ABB RobotStudio station: Sixth Assignment.rspag

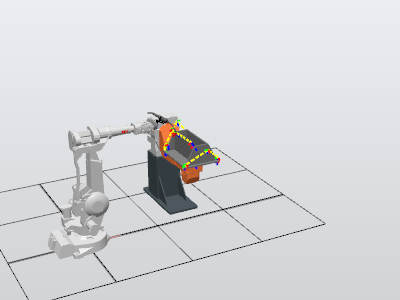
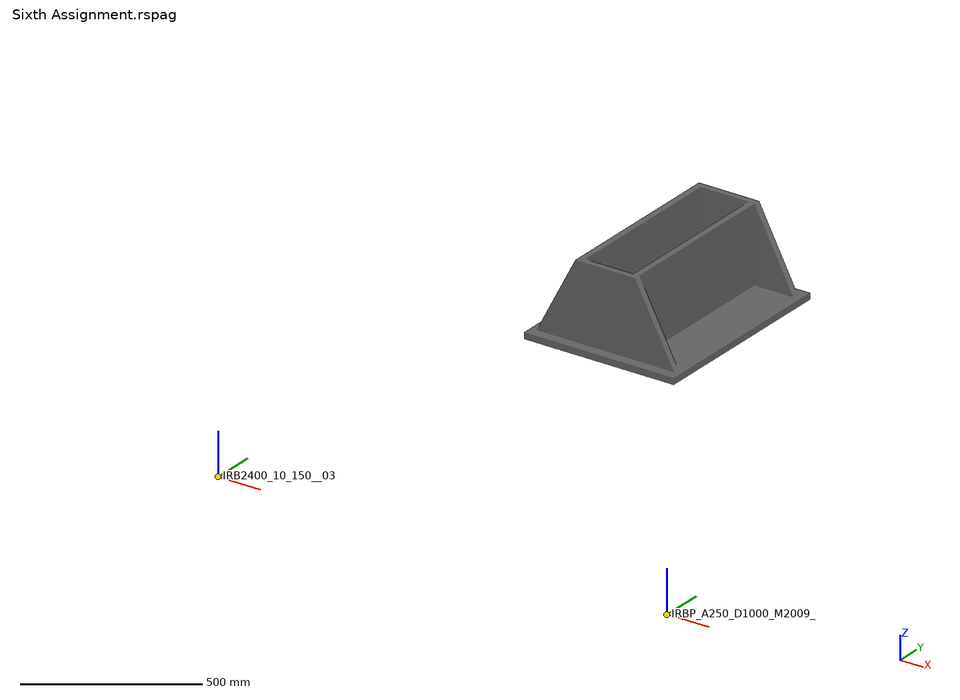
[picture v1: parts stored in the station drawn from their meshes, with robot base, taught points and paths (robot models come from the ABB library and are not in the file)]
--- station ---
Station station (saved by RobotStudio 24.1.10713.1)
Controller Controller
  mechanical unit ROB_1: IRB2400_10_150__03, 6 joints, base frame (0, 0, 0) mm
  mechanical unit STN1: IRBP_A250_D1000_M2009_REV1_01, 2 joints, base frame (0, 0, 0) mm
Layout (positions relative to the parent item):
  - IRB2400_10_150__03 [mechanism, from %ABB.RobotStudio.Models.IRB2400%\IRB2400_10_150_G_03.rslib] at (0, 0, 0) mm; joint values [0, 0.0266, 0.0287, -3.1416, -0.0726, 3.1416] (rad or m)
  - AW_Gun_PSF_25 [mechanism, from %ABB.RobotStudio.Models.ArcWelding%\AW_Gun_PSF_25.rslib] at (961.88, 0, 1424.46) mm, rotated rx 180 ry 84.2 rz 180 deg
  - IRBP_A250_D1000_M2009_REV1_01 [mechanism] at (1500, 0, 0) mm, rotated rx 0 ry 0 rz 90 deg; joint values [0, 0] (rad or m)
      links: Base, Link1, Link2
  - weldpiece [part] at (1500, 0, 900) mm, rotated rx 0 ry 0 rz -90 deg, size 650 x 500 x 270 mm
Attachment: AW_Gun_PSF_25 is attached to IRB2400_10_150__03 / Link6
Attachment: weldpiece is attached to IRBP_A250_D1000_M2009_REV1_01 / Link2

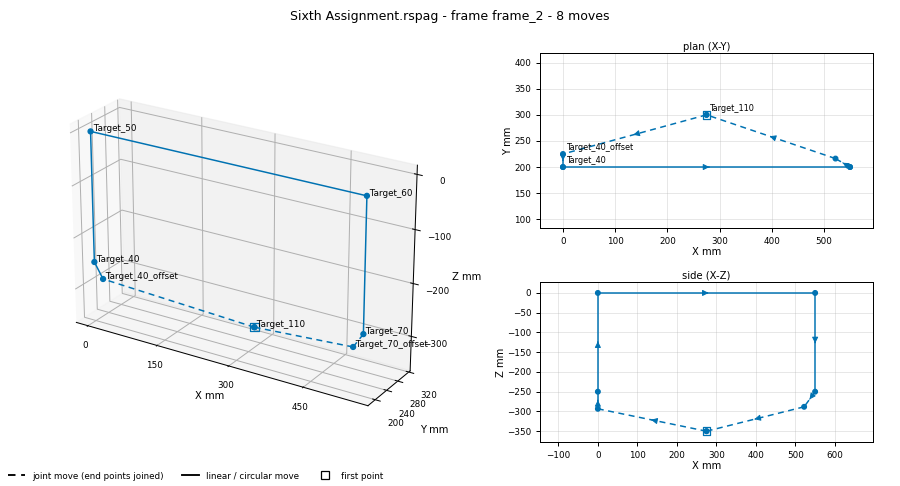
[picture p0: tool path of Sixth Assignment.rspag in frame frame_2, 8 of 20 moves have a stored position in this frame; points joined in program order, loops and branches not executed]
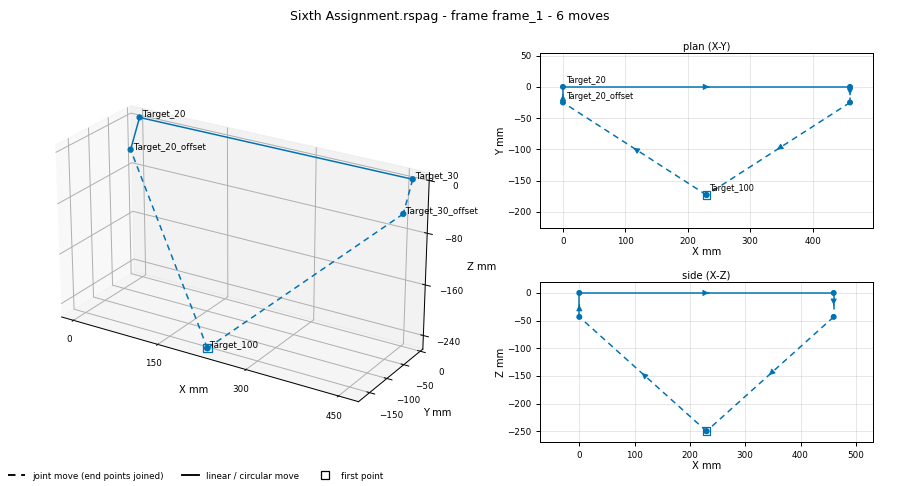
[picture p1: tool path of Sixth Assignment.rspag in frame frame_1, 6 of 20 moves have a stored position in this frame; points joined in program order, loops and branches not executed]
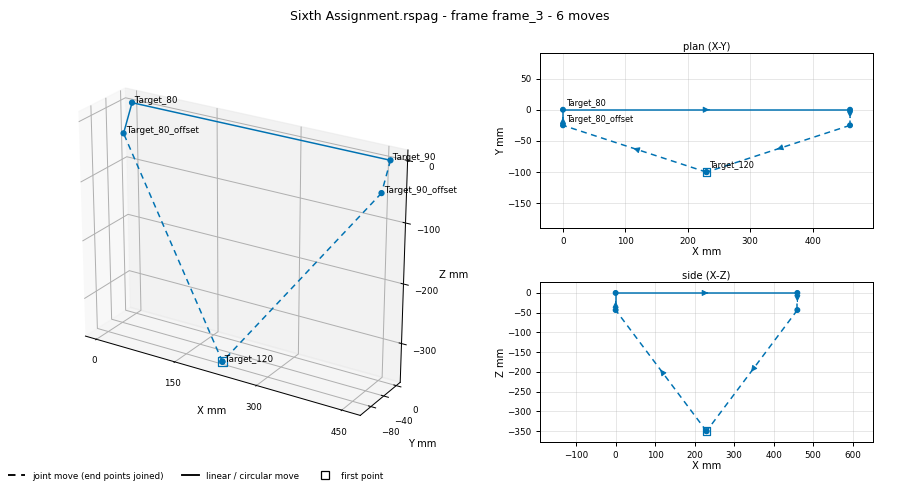
[picture p2: tool path of Sixth Assignment.rspag in frame frame_3, 6 of 20 moves have a stored position in this frame; points joined in program order, loops and branches not executed]
--- Backups/Controller/RAPID/TASK1/PROGMOD/CalibData.mod ---
MODULE CalibData
    PERS tooldata AW_Gun:=[TRUE,[[119.5,0,352],[0.890213743,0,0.455543074,0]],[1,[0,0,100],[1,0,0,0],0,0,0]];
    TASK PERS wobjdata frame_1:=[FALSE,FALSE,"STN1",[[0,0,0],[1,0,0,0]],[[295,230,20],[0,-0.707106781,0.707106781,0]]];
    TASK PERS wobjdata frame_2:=[FALSE,FALSE,"STN1",[[0,0,0],[1,0,0,0]],[[-275,100,20],[0,1,0,0]]];
    TASK PERS wobjdata frame_3:=[FALSE,FALSE,"STN1",[[0,0,0],[1,0,0,0]],[[-295,-230,20],[0,0.707106781,0.707106781,0]]];
ENDMODULE

--- Backups/Controller/RAPID/TASK1/PROGMOD/Module1.mod ---
MODULE Module1
    CONST robtarget Target_10:=[[1173.703101454,0,1133.009964248],[0.050594997,0,0.998719253,0],[0,0,0,0],[9E+09,9E+09,9E+09,9E+09,9E+09,9E+09]];
    CONST robtarget Target_20:=[[0,0,0],[0.683012702,-0.183012702,-0.183012702,-0.683012702],[-1,-1,0,0],[9E+09,0,-90,9E+09,9E+09,9E+09]];
    CONST robtarget Target_20_offset:=[[0,-25.000000009,-43.301270184],[0.683012702,-0.183012702,-0.183012702,-0.683012702],[-1,-1,0,0],[9E+09,0,-90,9E+09,9E+09,9E+09]];
    CONST robtarget Target_30:=[[460,0,0],[0.683012702,-0.183012702,-0.183012702,-0.683012702],[0,0,-1,0],[9E+09,0,-90,9E+09,9E+09,9E+09]];
    CONST robtarget Target_30_offset:=[[460,-25.000000009,-43.301270184],[0.683012702,-0.183012702,-0.183012702,-0.683012702],[0,0,-1,0],[9E+09,0,-90,9E+09,9E+09,9E+09]];
    CONST robtarget Target_100:=[[230,-173.205080735,-249.999999963],[0.683012702,-0.183012702,-0.183012702,-0.683012702],[0,0,-1,0],[9E+09,0,-90,9E+09,9E+09,9E+09]];

    CONST robtarget Target_40:=[[0,200,-250],[0.683012702,0.183012702,-0.183012702,0.683012702],[0,-2,1,0],[9E+09,0,0,9E+09,9E+09,9E+09]];
    CONST robtarget Target_40_offset:=[[0,225.000000009,-293.301270184],[0.683012702,0.183012702,-0.183012702,0.683012702],[0,-1,0,0],[9E+09,0,0,9E+09,9E+09,9E+09]];
    CONST robtarget Target_50:=[[0,200,0],[0.683012702,0.183012702,-0.183012702,0.683012702],[0,-2,1,0],[9E+09,0,0,9E+09,9E+09,9E+09]];
    CONST robtarget Target_60:=[[550,200,0],[0.470811924,0.342985757,-0.000965614,0.812832067],[0,-2,1,0],[9E+09,0,0,9E+09,9E+09,9E+09]];
    CONST robtarget Target_70:=[[550,200,-250],[0.470811924,0.342985757,-0.000965614,0.812832067],[0,-2,0,0],[9E+09,0,0,9E+09,9E+09,9E+09]];
    CONST robtarget Target_70_offset:=[[522.166480045,216.226666637,-288.235983795],[0.470811924,0.342985757,-0.000965614,0.812832067],[0,-2,0,0],[9E+09,0,0,9E+09,9E+09,9E+09]];
    CONST robtarget Target_110:=[[275,300,-350],[0.683012702,0.183012702,-0.183012702,0.683012702],[0,-2,0,0],[9E+09,0,0,9E+09,9E+09,9E+09]];

    CONST robtarget Target_80_offset:=[[0,-25.000000009,-43.301270184],[0.683012702,-0.183012702,-0.183012702,-0.683012702],[0,0,0,0],[9E+09,0,90,9E+09,9E+09,9E+09]];
    CONST robtarget Target_80:=[[0,0,0],[0.683012702,-0.183012702,-0.183012702,-0.683012702],[0,0,0,0],[9E+09,0,90,9E+09,9E+09,9E+09]];
    CONST robtarget Target_90:=[[460,0,0],[0.683012702,-0.183012702,-0.183012702,-0.683012702],[0,0,0,0],[9E+09,0,90,9E+09,9E+09,9E+09]];
    CONST robtarget Target_90_offset:=[[460,-25.000000009,-43.301270184],[0.683012702,-0.183012702,-0.183012702,-0.683012702],[0,0,0,0],[9E+09,0,90,9E+09,9E+09,9E+09]];
    CONST robtarget Target_120:=[[230,-100,-350],[0.683012702,-0.183012702,-0.183012702,-0.683012702],[0,0,0,0],[9E+09,0,90,9E+09,9E+09,9E+09]];
!***********************************************************
    !
    ! Module:  Module1
    !
    ! Description:
    !   <Insert description here>
    !
    ! Author: haba0028
    !
    ! Version: 1.0
    !
    !***********************************************************


    !***********************************************************
    !
    ! Procedure main
    !
    !   This is the entry point of your program
    !
    !***********************************************************
    PROC main()
        !Add your code here
        WaitTime 0.3;
        Path_10;
        WaitTime 0.3;
        Path_30;
        WaitTime 0.3;
        Path_20;
    ENDPROC
    PROC Path_10()
        ActUnit STN1;
        MoveJ Target_100,v200,fine,AW_Gun\WObj:=frame_1;
        MoveJ Target_20_offset,v200,fine,AW_Gun\WObj:=frame_1;
        MoveL Target_20,v200,fine,AW_Gun\WObj:=frame_1;
        MoveL Target_30,v200,fine,AW_Gun\WObj:=frame_1;
        MoveJ Target_30_offset,v200,fine,AW_Gun\WObj:=frame_1;
        MoveJ Target_100,v200,fine,AW_Gun\WObj:=frame_1;
        DeactUnit STN1;
    ENDPROC
    PROC Path_20()
        ActUnit STN1;
        MoveJ Target_110,v200,fine,AW_Gun\WObj:=frame_2;
        MoveJ Target_40_offset,v200,fine,AW_Gun\WObj:=frame_2;
        MoveL Target_40,v200,fine,AW_Gun\WObj:=frame_2;
        MoveL Target_50,v200,fine,AW_Gun\WObj:=frame_2;
        MoveL Target_60,v200,fine,AW_Gun\WObj:=frame_2;
        MoveL Target_70,v200,fine,AW_Gun\WObj:=frame_2;
        MoveJ Target_70_offset,v200,fine,AW_Gun\WObj:=frame_2;
        MoveJ Target_110,v200,fine,AW_Gun\WObj:=frame_2;
        DeactUnit STN1;
    ENDPROC
    PROC Path_30()
        ActUnit STN1;
        MoveJ Target_120,v200,fine,AW_Gun\WObj:=frame_3;
        MoveJ Target_80_offset,v200,fine,AW_Gun\WObj:=frame_3;
        MoveL Target_80,v200,fine,AW_Gun\WObj:=frame_3;
        MoveL Target_90,v200,fine,AW_Gun\WObj:=frame_3;
        MoveJ Target_90_offset,v200,fine,AW_Gun\WObj:=frame_3;
        MoveJ Target_120,v200,fine,AW_Gun\WObj:=frame_3;
        DeactUnit STN1;
    ENDPROC
ENDMODULE

--- Backups/Controller/SYSPAR/EIO.cfg ---
EIO:CFG_1.0:6:1::
#
INDUSTRIAL_NETWORK:

      -Name "PROFIBUS" -Label "PROFIBUS Controller Network"\
      -CfgPath "HOME/pbus_cfg.bin"
#
LOCAL_DEVICE:

      -Name "DRVIO_1" -Network "Local" -StateWhenStartup "Deactivated"\
      -TrustLevel "DRVIO_TRUSTLEVEL"
#
EIO_CROSS:

      -Name "Cross_doACT_K1" -Res "doACT_K1" -Act1 "soACT_STN1"

      -Name "Cross_doACT_K3" -Res "doACT_K3" -Act1 "soACT_STN1"

      -Name "Cross_siSTN1_ACT" -Res "siSTN1_ACT" -Act1 "diK1_ACT" -Oper1 "AND"\
      -Act2 "diK3_ACT"

      -Name "Cross_doACT_K11" -Res "doACT_K11" -Act1 "doACT_K13"
#
EIO_DEVICE_TRUSTLEVEL:

      -Name "DRVIO_TRUSTLEVEL" -ActionWhenLost "NONE" -ReportWhenLost "NONE"\
      -ReportWhenReconnected "NONE"
#
EIO_SIGNAL:

      -Name "doACT_K1" -SignalType "DO" -Device "DRVIO_1" -DeviceMap "0"

      -Name "doACT_K3" -SignalType "DO" -Device "DRVIO_1" -DeviceMap "2"

      -Name "doACT_K11" -SignalType "DO" -Device "DRVIO_1" -DeviceMap "5"

      -Name "doACT_K13" -SignalType "DO" -Device "DRVIO_1" -DeviceMap "7"

      -Name "diK1_ACT" -SignalType "DI" -Device "DRVIO_1" -DeviceMap "0"\
      -FiltPas 50 -FiltAct 50

      -Name "diK3_ACT" -SignalType "DI" -Device "DRVIO_1" -DeviceMap "2"\
      -FiltPas 50 -FiltAct 50

      -Name "soACT_STN1" -SignalType "DO" -DeviceMap "0"

      -Name "siSTN1_ACT" -SignalType "DI" -DeviceMap "0"
